(* CODESYS project SNDLTN_Hestia.library
   Company: Sandolution
   Title: SNDLTN_Hestia
   Description: Library in to aid setting up an automated domotica system.
   Author: S. Verbeek
   Version: 1.1.200929

Project tree, tasks and I/O mapping:
  libraries: StringUtils, * (System); Standard, * (System); CAA Real Time Clock Extern, * (CAA Technical Workgroup); SysSocket, * (System); CAA Net Base Services, * (CAA Technical Workgroup); SysTypes Interfaces, * (System); CmpErrors Interfaces, * (System); CAA Types, 3.0.0.2 (3S - Smart Software Solutions GmbH); CAA Tick, 3.0.0.0 (3S - Smart Software Solutions GmbH)
  Constants/
    global variables Hestia_Constants
    global variables Hestia_Properties
  Enums/
    data type Hestia_eAlarmHandler_Category
    data type Hestia_eAlarmHandler_Severity
    data type Hestia_eInputMode
    data type Hestia_eWeekday
    data type Hestia_eAlarmHandler_Sorting
  Function Blocks/
    Alarms/
      function block Hestia_AlarmHandler [ST]: Main, ShiftOutput
      function block Hestia_AlarmMessager [ST]: Main
    Colors/
      function block Hestia_Fader [ST]: Main
    Heating/
      function block Hestia_TemperatureController [ST]: Main
    Time/
      function block Hestia_WeekClock [ST]: Main, CheckWeekday
      function block Hestia_TONR [ST]: Main
    Network/
      function block Hestia_Pinger [ST]: Main
    I/O-Digital/
      function block Hestia_OutputDelay [ST]: Main
      function block Hestia_OutputHistory [ST]: Main
      function block Hestia_InputClicks [ST]: Main
      function block _Hestia_Template_xInxInvert_xOut [ST]: Main
      function block Hestia_PulseWidthModulation [ST]: Main
      function block Hestia_StateFilter [ST]: Main
    I/O-Analog/
      function block Hestia_ArrayAverage [ST]: Main
      function block Hestia_SwitchPoint_Single [ST]: Main
      function block Hestia_MovingAverage [ST]: Main
  Structs/
    data type Hestia_scWeekClockEntry
    data type Hestia_scAlarmHandler_Entry
  Variables/
  Visualizations/
  text list GlobalTextList
  program ChangeLog [ST]
  Functions/
    function Hestia_DateToWeekday [ST]
    function Hestia_ReplaceChars [ST]
    function Hestia_RandomValue [ST]
*)

// Enums/Hestia_eAlarmHandler_Category
{attribute 'qualified_only'}
{attribute 'strict'}
{attribute 'to_string'}
TYPE Hestia_eAlarmHandler_Category :
(
	System := 0,
	Security,
	Network,
	Weather,
	Climate,
	Devices,
	Monitoring
);
END_TYPE

// Enums/Hestia_eAlarmHandler_Severity
{attribute 'qualified_only'}
{attribute 'to_string'}
TYPE Hestia_eAlarmHandler_Severity :
(
	_0_Debug := 0,			//Debugging output - use only for debugging
	_1_Informational,		//Normal info for user - not important
	_2_Notice,				//Important info for user 
	_3_Warning,				 //Warning occured - attention required
	_4_Error,				//Error occured, continue processing - attention required
	_5_Critical,			//Cricital error which could comprimise functionality - action required
	_6_Alert,				//Inmediate action required to prevent further damage
	_7_Emergency			//System unusable / panic
);
END_TYPE

// Structs/Hestia_scWeekClockEntry
TYPE Hestia_scWeekClockEntry :
STRUCT
	//Week
	eWeekday					: Hestia_eWeekday;	//Individual bits also usable
	
	//Time on which output is on
	todSwitchPoint_On			: TIME_OF_DAY;		//On
	todSwitchPoint_Off			: TIME_OF_DAY;		//Off
	
	//Custom
	dwCustomAction				: DWORD;			//Specify your own custom action here, defined as number
END_STRUCT
END_TYPE

// Enums/Hestia_eInputMode
{attribute 'qualified_only'}
{attribute 'strict'}
TYPE Hestia_eInputMode :
(
	STATE := 0,
	RISING_EDGE,
	FALLING_EDGE
);
END_TYPE

// Enums/Hestia_eWeekday
{attribute 'qualified_only'}
{attribute 'to_string'}
TYPE Hestia_eWeekday :
(
	Sunday := 1,
	Monday := 2,
	Tuesday := 4,
	Wednesday := 8,
	Thursday := 16,
	Friday := 32,
	Saturday := 64,
	MonTueWedThuFri := 62,
	SatSun := 65,
	All	:= 127
) WORD;	//Set type WORD
END_TYPE

// Structs/Hestia_scAlarmHandler_Entry
TYPE Hestia_scAlarmHandler_Entry :
STRUCT
	xActive			:BOOL;
	xAckNeeded		:BOOL;
	wErrorCode		:WORD;
	eSeverity		:Hestia_eAlarmHandler_Severity;
	eCategory		:Hestia_eAlarmHandler_Category;
	sText			:STRING(Hestia_Properties.uiAlarmHandler_StringSize) := '';
END_STRUCT
END_TYPE

// Enums/Hestia_eAlarmHandler_Sorting
{attribute 'qualified_only'}
{attribute 'strict'}
TYPE Hestia_eAlarmHandler_Sorting :
(
	NoSorting := 0,
	Severity,
	TimeStamp_Oldest,
	TimeStamp_Newest
);
END_TYPE

// Constants/Hestia_Constants
{attribute 'qualified_only'}
VAR_GLOBAL CONSTANT
	uiAlarmHandler_Severity	: UINT := 8; //(0-7)
END_VAR

// Constants/Hestia_Properties
{attribute 'qualified_only'}
{attribute 'strict'}
VAR_GLOBAL CONSTANT
	uiAlarmHandler_Inputs					: UINT := 64;
	uiAlarmHandler_StringSize				: UINT := 128;
	uiAlarmHandler_Outputs					: UINT := 8;

	uiWeekClock_Entries						: UINT := 8;
	
	uiReplaceChars_StringSize				: UINT := 128;
	
	uiPinger_Samples						: UINT := 4;
	
	uiStateFilter_Inputs					: UINT := 8;
END_VAR

// ChangeLog
PROGRAM ChangeLog
VAR
END_VAR

//Library in extension to SNDLTN_Domoticz library.
//Contains functions for setting up a domotics system.

//V1.1.200929
//Fixed small bug in Switchpoint Single where hysteresis didn't work when inverted.
//Added PulseWidthModulation to control outputs.

//V1.1.200612
//Added Hestia_Pinger for ICMP pinging of network slaves
//Adjusted Hestia_ReplaceChars so it supports up to 8 chars instead of 1

//V1.1.200226
//Rewrote AlarmHandler for better sorting and handling of alarms.
//Added implementation of AlarmNotifier to send messages from the alarm handler
//Fixed bug in WeekClock on which wrong day was used for setpoints on/off spread across two days.

//V1.1.200125
//Upgraded to CoDeSys verison 3.5.14.40.
//Changed HeatingControl to TemperatureControl.

//V1.1.191207
//Added implementation of WeekClock.
//Added hysteresis to HeatingControl

//V1.1.191101:
//Added HeatingControl for simple control of heating systems.

//V1.1 - Okt 2019:
//Extension of OutputDelay and OutputHistory with eInputMode to select behaviour for different sensor types.
//Fixed bug of ColorFade where wrong constant was used. Also changed implementation to use 1..Constant instead of 0..Constant-1.

//V1.0 - Aug 2019:
//Implementation of AlarmHandler, InputClicks, OutputDelay, OutputHistory and ArrayAverage
//Sep 2019:
//Implementation of ColorFade

END_PROGRAM

// Function Blocks/Network/Hestia_Pinger
{attribute 'conditionalshow_all_locals'}
FUNCTION_BLOCK Hestia_Pinger
VAR_INPUT
	sIPAdress			:STRING := '192.168.1.1';
	udTimeOut			:UDINT := 100;
END_VAR             	 
VAR_OUTPUT          	 
	xAlive				:BOOL;
	udReplyTime			:UDINT;
END_VAR             	 
VAR                 	 
	ascResult			:ARRAY[1..Hestia_Properties.uiPinger_Samples] OF RTS_IEC_RESULT;
	rAlive_avg			:REAL;
	audReplyTime		:ARRAY[1..Hestia_Properties.uiPinger_Samples] OF UDINT;
	rReplyTime_avg		:REAL;
	SysException		:__SYSTEM.ExceptionCode;
	uiSamplesTaken		:UINT;
	idx					:INT;
END_VAR

Main();

ACTION Main:
{attribute 'conditionalshow'}
__TRY
	uiSamplesTaken := 1;
	
	IF Hestia_Properties.uiPinger_Samples > 0 THEN
		//Take all samples
		WHILE uiSamplesTaken <= Hestia_Properties.uiPinger_Samples DO
			//Get result and put in array
			ascResult[uiSamplesTaken] := SysSockPing(szIPAddress:= sIPAdress, ulTimeout:= udTimeOut, pulReplyTime:= ADR(audReplyTime[uiSamplesTaken]));
			
			//Go to next sample
			uiSamplesTaken := uiSamplesTaken + 1;
		
		END_WHILE
		
		rAlive_avg := 0;
		rReplyTime_avg := 0;
		
		FOR idx := 1 TO TO_INT(Hestia_Properties.uiPinger_Samples) DO
			//Only count valid responds, all other means offline (ERR_TIMEOUT)
			IF ascResult[idx] = CmpErrors.Errors.ERR_OK THEN
				rAlive_avg := rAlive_avg + 1;
			END_IF
			
			//Add timeout
			rReplyTime_avg := rReplyTime_avg + TO_REAL(audReplyTime[idx]);

		END_FOR
		
		//Calculate averages
		xAlive := (rAlive_avg/Hestia_Properties.uiPinger_Samples) > 0;	//One of the samples is set to true
		udReplyTime := TO_UDINT(rReplyTime_avg/Hestia_Properties.uiPinger_Samples);
		
	END_IF
	
__CATCH(SysException)
	;
__ENDTRY
END_ACTION

END_FUNCTION_BLOCK

// Functions/Hestia_ReplaceChars
FUNCTION Hestia_ReplaceChars : STRING(Hestia_Properties.uiReplaceChars_StringSize);
VAR_INPUT
	sInput			: STRING(Hestia_Properties.uiReplaceChars_StringSize);
	sCharFind		: STRING(16);
	sCharReplace	: STRING(16);
END_VAR
VAR
	iSearchPos		: INT;
	iReplaceFind	: INT;	//Check if replace string contains find string
	idx				: WORD;
END_VAR

IF sInput <> ''
AND sCharFind <> '' THEN
//AND sCharReplace <> '' THEN
	iSearchPos := 0;
	Hestia_ReplaceChars := sInput;
	
	iReplaceFind := StrFindA( ADR(sCharReplace),							//pst1
							ADR(sCharFind),									//pst2
							0);												//uiSearchStart

	FOR idx := 0 TO Hestia_Properties.uiReplaceChars_StringSize DO
		iSearchPos := StrFindA( ADR(Hestia_ReplaceChars),					//pst1
								ADR(sCharFind),								//pst2
								TO_UINT(iSearchPos));						//uiSearchStart
	
		IF iSearchPos <> 0 THEN						
			StrReplaceA(ADR(Hestia_ReplaceChars),							//pstInput
						SIZEOF(Hestia_ReplaceChars),						//uiInputBufferSize
						ADR(sCharReplace),									//pstReplaceWith
						LEN(Hestia_ReplaceChars),							//iLengthInput
						LEN(sCharFind),										//iLengthToReplace
						LEN(sCharReplace),									//iLengthToReplaceWith
						iSearchPos);										//iPosition
			iSearchPos := iSearchPos + iReplaceFind;
		ELSE
			EXIT;
		END_IF
	END_FOR
	
END_IF

END_FUNCTION

// Function Blocks/I/O-Digital/Hestia_OutputDelay
{attribute 'conditionalshow_all_locals'}
//Delay an output signal by x time
//Individual outputs are set active after set time and are reset again after the set time has passed.
//For example: 1 minut output is set after 1 minute high signal, and reset 1 minute after low signal.
FUNCTION_BLOCK Hestia_OutputDelay EXTENDS _Hestia_Template_xInxInvert_xOut
VAR_OUTPUT
	xOut_1, xOut_5, xOut_15, xOut_30, xOut_60		:BOOL;	//Input status 1/5/15/30/60m ago
END_VAR
VAR
	TON_1M, TON_5M, TON_15M, TON_30M, TON_60M		:TON;
	TOF_1M, TOF_5M, TOF_15M, TOF_30M, TOF_60M		:TOF;
END_VAR

Main();

ACTION Main:
{attribute 'conditionalshow'}
//Call parent
SUPER^.Main();

//Timed outputs
TON_1M(	IN:=xIn_int OR TOF_1M.Q, PT:=T#1M);
TOF_1M(	IN:=xIn_int AND TON_1M.Q, PT:=T#1M);
xOut_1 := TON_1M.Q OR TOF_1M.Q;

TON_5M(	IN:=xIn_int OR TOF_5M.Q, PT:=T#5M);
TOF_5M(	IN:=xIn_int AND TON_5M.Q, PT:=T#5M);
xOut_5 := TON_5M.Q OR TOF_5M.Q; 

TON_15M(IN:=xIn_int OR TOF_15M.Q, PT:=T#15M);
TOF_15M(IN:=xIn_int AND TON_15M.Q, PT:=T#15M);
xOut_15 := TON_15M.Q OR TOF_15M.Q; 

TON_30M(IN:=xIn_int OR TOF_30M.Q, PT:=T#30M);
TOF_30M(IN:=xIn_int AND TON_30M.Q, PT:=T#30M);
xOut_30 := TON_30M.Q OR TOF_30M.Q; 

TON_60M(IN:=xIn_int OR TOF_60M.Q, PT:=T#60M);
TOF_60M(IN:=xIn_int AND TON_60M.Q, PT:=T#60M);
xOut_60 := TON_60M.Q OR TOF_60M.Q;
END_ACTION

END_FUNCTION_BLOCK

// Function Blocks/I/O-Digital/_Hestia_Template_xInxInvert_xOut
{attribute 'conditionalshow'}
FUNCTION_BLOCK _Hestia_Template_xInxInvert_xOut
VAR_INPUT
	xIn			:BOOL;		//Input signal
	xInvert		:BOOL;		//Normally open / normally closed input
END_VAR
VAR_OUTPUT
	xOut		:BOOL;		//Direct output
END_VAR
VAR
	xIn_int		:BOOL;
END_VAR

//Main is called from extended slaves

ACTION Main:
//Input
xIn_int := xIn XOR xInvert;

//Direct output
xOut := xIn_int;
END_ACTION

END_FUNCTION_BLOCK

// Function Blocks/I/O-Digital/Hestia_OutputHistory
{attribute 'conditionalshow_all_locals'}
FUNCTION_BLOCK Hestia_OutputHistory EXTENDS _Hestia_Template_xInxInvert_xOut
VAR_INPUT
	eInputMode	:Hestia_eInputMode;		//Type of reaction to input
END_VAR
VAR_OUTPUT
	xOut_1, xOut_5, xOut_15, xOut_30, xOut_60		:BOOL;	//Input status 1/5/15/30/60m ago
END_VAR
VAR
	TOF_1M, TOF_5M, TOF_15M, TOF_30M, TOF_60M		:TOF;
	xIn_mode,xIn_old:BOOL;
END_VAR

Main();

ACTION Main:
{attribute 'conditionalshow'}
//Call parent
SUPER^.Main();

CASE eInputMode OF
	Hestia_eInputMode.STATE:	
		xIn_mode := xIn_int;
	
	Hestia_eInputMode.RISING_EDGE:	
		xIn_mode := xIn_int AND NOT xIn_old;
			
	Hestia_eInputMode.FALLING_EDGE:	
		xIn_mode := NOT xIn_int AND xIn_old;
END_CASE

//Save state
xIn_old := xIn_int;

//Timed outputs
TOF_1M(	IN:=xIn_mode, PT:=T#1M, Q => xOut_1);
TOF_5M(	IN:=xIn_mode, PT:=T#5M, Q => xOut_5);
TOF_15M(IN:=xIn_mode, PT:=T#15M, Q => xOut_15);
TOF_30M(IN:=xIn_mode, PT:=T#30M, Q => xOut_30);
TOF_60M(IN:=xIn_mode, PT:=T#60M, Q => xOut_60);
END_ACTION

END_FUNCTION_BLOCK

// Function Blocks/I/O-Digital/Hestia_InputClicks
{attribute 'conditionalshow_all_locals'}
FUNCTION_BLOCK Hestia_InputClicks EXTENDS _Hestia_Template_xInxInvert_xOut
VAR_INPUT
	tDebounce			:TIME := T#25MS;		//Debounce time
	tReset				:TIME := T#500MS;		//Reset outputs after set time
END_VAR
VAR_OUTPUT
	xOut_Pulse			:BOOL;
	xOut_PulseInv		:BOOL;
	xOut_Long			:BOOL;
	xOut_Single			:BOOL;
	xOut_Double			:BOOL;
	xOut_Triple			:BOOL;
END_VAR
VAR
	TON_Debounce		:TON;			//Filter input signal
	RTRIG_In			:R_TRIG;		//Pulse trigger
	FTRIG_In			:F_TRIG;		//Pulse trigger
	byCount				:BYTE;			//Count edges
	TON_Reset			:TON;			//Reset after time passed
END_VAR

Main();

ACTION Main:
{attribute 'conditionalshow'}
//Call parent
SUPER^.Main();

//Trigger on input
TON_Debounce(IN:=xIn_int, PT:=tDebounce);
RTRIG_In(CLK:=TON_Debounce.Q);
FTRIG_In(CLK:=TON_Debounce.Q);

//Count inputs
IF RTRIG_In.Q THEN
	byCount := byCount + 1;
END_IF

//Reset after set time, but reset timer each time input is received
TON_Reset(IN:=(byCount>0) AND NOT RTRIG_In.Q, PT:=tReset);
IF TON_Reset.Q AND NOT TON_Debounce.Q THEN
	byCount := 0;
END_IF

//Outputs
//xOut is written in template function 
xOut_Pulse 		:= RTRIG_In.Q;		//Single flank
xOut_PulseInv 	:= FTRIG_In.Q;		//Single flank inverted
xOut_Long 		:= TON_Debounce.Q AND TON_Reset.Q;	//Long press
xOut_Single 	:= (byCount = 1);	//1
xOut_Double 	:= (byCount = 2);	//2
xOut_Triple 	:= (byCount = 3);	//3
END_ACTION

END_FUNCTION_BLOCK

// Function Blocks/I/O-Analog/Hestia_ArrayAverage
{attribute 'conditionalshow_all_locals'}
FUNCTION_BLOCK Hestia_ArrayAverage
VAR_INPUT
	arValues		:ARRAY[1..iSamples] OF REAL := [iSamples(-999)];
END_VAR
VAR_OUTPUT
	rValue_AVG		:REAL;
END_VAR
VAR
	byX				:BYTE;
	byCnt			:BYTE;
END_VAR
VAR CONSTANT
	iSamples		:INT := 8;
END_VAR

Main();

ACTION Main:
{attribute 'conditionalshow'}
//Reset
rValue_AVG := 0;
byCnt := 0;

//Valid values
//Add all values
FOR byX := 1 TO TO_BYTE(iSamples) DO
	IF arValues[byX] <> -999 THEN
		byCnt := byCnt + 1;
		rValue_AVG := rValue_AVG + arValues[byX];
	END_IF
END_FOR

//Calc average
IF byCnt <> 0 THEN
	rValue_AVG := rValue_AVG / byCnt;
ELSE
	rValue_AVG := 0.0;
END_IF
END_ACTION

END_FUNCTION_BLOCK

// Function Blocks/Heating/Hestia_TemperatureController
{attribute 'conditionalshow_all_locals'}
FUNCTION_BLOCK Hestia_TemperatureController
VAR_INPUT
	
	rTemperature_Actual		:REAL;			//Actual room temperature (might be altered by other functions already)
	rTemperature_Hysteresis :REAL;			//Hysteresis
	
	rTemperature_Setpoint	:REAL;			//Setpoint for control
	
	xOverride				:BOOL;			//Overrule setpoint + hysteresis
	rTemperature_Override	:REAL;			//Temperature override
                             
END_VAR                      
VAR_OUTPUT	 
	xCooling				:BOOL;			//Cooling should be activate                
	xHeating				:BOOL;			//Heating should be activate
	rTemperature_Out		:REAL;			//System setpoint
END_VAR                      
VAR                          
	xActBelowHysteresis		:BOOL;
	xActAboveHysteresis		:BOOL;
END_VAR

//Call main function
Main();

ACTION Main:
{attribute 'conditionalshow'}

//Below upper hysteresis limit
//Passing from below lower hysteresis limit
IF rTemperature_Actual < rTemperature_Setpoint
AND NOT xActAboveHysteresis
AND xActBelowHysteresis THEN
	xCooling := FALSE;
	xHeating := TRUE;

//Above upper hysteresis limit
ELSIF rTemperature_Actual >= rTemperature_Setpoint THEN
	xActAboveHysteresis := TRUE;
	xActBelowHysteresis := FALSE;
	xCooling := TRUE;
	xHeating := FALSE;

//Above lower hysteresis limit
//Passing from above higher hysteresis limit
ELSIF rTemperature_Actual >= (rTemperature_Setpoint - rTemperature_Hysteresis)
AND xActAboveHysteresis
AND NOT xActBelowHysteresis THEN
	xCooling := TRUE;
	xHeating := FALSE;
	
//Below lower hysteresis limit
ELSIF rTemperature_Actual < (rTemperature_Setpoint - rTemperature_Hysteresis) THEN
	xActAboveHysteresis := FALSE;
	xActBelowHysteresis := TRUE;
	xCooling := FALSE;
	xHeating := FALSE;

//Catch
ELSE
	xCooling := FALSE;
	xHeating := FALSE;	
END_IF
	
//Override active
IF xOverride THEN
	rTemperature_Out := rTemperature_Override;	
//Normal operation
ELSE
	rTemperature_Out := rTemperature_Setpoint;
END_IF
END_ACTION

END_FUNCTION_BLOCK

// Functions/Hestia_DateToWeekday
{attribute 'conditionalshow_all_locals'}
FUNCTION Hestia_DateToWeekday : Hestia_eWeekday
VAR_INPUT
	dDate				:DATE;	//Date to convert
END_VAR 
VAR
	sDate				:STRING(12);
	iYear,iMonth,iDay	:INT;
	iYearDigit,iCentury	:INT;
	iCalculate			:INT;
END_VAR

//Conversion is done using the Key Value method

//Convert to STRING and get INT values
sDate 		:= TO_STRING(dDate);
iYear 		:= TO_INT(MID(sDate,4,3));	//Extract length 4 from pos 3 (1970)
iYearDigit 	:= TO_INT(MID(sDate,2,5));	//Extract length 2 from pos 5 (70)
iCentury 	:= TO_INT(MID(sDate,2,3));	//Extract length 2 from pos 3 (19)
iMonth 		:= TO_INT(MID(sDate,2,8));	//Extract length 2 from pos 8 (01)
iDay 		:= TO_INT(MID(sDate,2,11));	//Extract length 2 from pos 11 (01)

//Take last two digits of the year and divide by 4, drop remainder
iCalculate 	:= iYearDigit / 4;
//Add day of month
iCalculate 	:=  iCalculate + iDay;
//Add key value
CASE iMonth OF
	1:	iCalculate := iCalculate + 1;
	2:	iCalculate := iCalculate + 4;
	3:	iCalculate := iCalculate + 4;
	4:	iCalculate := iCalculate + 0;
	5:	iCalculate := iCalculate + 2;
	6:	iCalculate := iCalculate + 5;
	7:	iCalculate := iCalculate + 0;
	8:	iCalculate := iCalculate + 3;
	9:	iCalculate := iCalculate + 6;
	10:	iCalculate := iCalculate + 1;
	11:	iCalculate := iCalculate + 4;
	12:	iCalculate := iCalculate + 6;
END_CASE
//Substract 1 for Jan/Feb if leap year
IF ((iYear MOD 4) = 0) AND (iMonth = 1 OR iMonth = 2) THEN
	iCalculate := iCalculate - 1;
END_IF
//Add century code
//Note that this only works from 1900 to 2100, date type doesn't support other centuries
CASE iCentury OF
	19:	iCalculate := iCalculate + 0;
	20:	iCalculate := iCalculate + 6;
	21:	iCalculate := iCalculate + 4;
END_CASE
//Add year digits
iCalculate := iCalculate + iYearDigit;
//Devide by 7 and take remainder
iCalculate := iCalculate MOD 7;
//Fix if 0, this is also saturday
IF iCalculate = 0 THEN
	iCalculate := 7;
END_IF
//Output
Hestia_DateToWeekday := TO_WORD(iCalculate);

END_FUNCTION

// Function Blocks/Time/Hestia_WeekClock
{attribute 'conditionalshow_all_locals'}
FUNCTION_BLOCK Hestia_WeekClock
VAR_INPUT
	xEnable					: BOOL;
	dtActDateTime			: DATE_AND_TIME;
	ascWeekClock_Entries	: ARRAY[1..Hestia_Properties.uiWeekClock_Entries] OF Hestia_scWeekClockEntry;
END_VAR
VAR_OUTPUT
	byEntryActive			: BYTE;
	dwAction				: DWORD;
END_VAR
VAR
	idx						: WORD;
	axSaveNextDay			: ARRAY[1..Hestia_Properties.uiWeekClock_Entries] OF BOOL;
END_VAR

Main();

ACTION Main:
{attribute 'conditionalshow'}

//Reset outputs
byEntryActive := 0;
dwAction := 0;

IF xEnable THEN
	
	//Loop all entries
	FOR idx := 1 TO Hestia_Properties.uiWeekClock_Entries DO
		
		//Check if entries are valid
		IF ascWeekClock_Entries[idx].todSwitchPoint_On <> TOD#00:00:00
		AND ascWeekClock_Entries[idx].todSwitchPoint_Off <> TOD#00:00:00
		AND ascWeekClock_Entries[idx].todSwitchPoint_On <> ascWeekClock_Entries[idx].todSwitchPoint_Off THEN
		
			//Time on/off lays in the same day and in correct order
			IF ascWeekClock_Entries[idx].todSwitchPoint_On < ascWeekClock_Entries[idx].todSwitchPoint_Off THEN
			
				//Actual time within range of setpoints
				IF TO_TOD(dtActDateTime) >= ascWeekClock_Entries[idx].todSwitchPoint_On
				AND TO_TOD(dtActDateTime) < ascWeekClock_Entries[idx].todSwitchPoint_Off
				//Correct day active
				AND CheckWeekday(TO_DATE(dtActDateTime), ascWeekClock_Entries[idx].eWeekday, FALSE) THEN
					byEntryActive := TO_BYTE(idx);
					dwAction := ascWeekClock_Entries[idx].dwCustomAction;
				END_IF	
				
			//Time on/off lay on two different days. Use weekday of ON switchpoint
			ELSIF ascWeekClock_Entries[idx].todSwitchPoint_On > ascWeekClock_Entries[idx].todSwitchPoint_Off THEN
				//Actual time within range of setpoints
				IF (TO_TOD(dtActDateTime) >= ascWeekClock_Entries[idx].todSwitchPoint_On
					OR (TO_TOD(dtActDateTime) < ascWeekClock_Entries[idx].todSwitchPoint_Off AND axSaveNextDay[idx]))
				AND (TO_TOD(dtActDateTime) < ascWeekClock_Entries[idx].todSwitchPoint_Off 
					OR (TO_TOD(dtActDateTime) >= ascWeekClock_Entries[idx].todSwitchPoint_On AND (TO_TOD(dtActDateTime) <= TOD#23:59:59)))
				//Correct day active
				AND (CheckWeekday(TO_DATE(dtActDateTime), ascWeekClock_Entries[idx].eWeekday, TRUE) OR axSaveNextDay[idx]) THEN
					axSaveNextDay[idx] := TRUE;
					byEntryActive := TO_BYTE(idx);
					dwAction := ascWeekClock_Entries[idx].dwCustomAction;
				ELSE
					axSaveNextDay[idx] := FALSE;
				END_IF	
			END_IF
			
		END_IF
	
	END_FOR

END_IF
END_ACTION

METHOD CheckWeekday : BOOL
VAR_INPUT
	dActDate	: DATE;
	eWeekday	: Hestia_eWeekday;
	xDayInPast	: BOOL;
END_VAR
CheckWeekday := 
			//Check current day (setpoints on same day)
			(NOT xDayInPast
			AND ((Hestia_DateToWeekday(dActDate) = 1 AND eWeekday.0)
			OR (Hestia_DateToWeekday(dActDate) = 2 AND eWeekday.1)
			OR (Hestia_DateToWeekday(dActDate) = 3 AND eWeekday.2)
			OR (Hestia_DateToWeekday(dActDate) = 4 AND eWeekday.3)
			OR (Hestia_DateToWeekday(dActDate) = 5 AND eWeekday.4)
			OR (Hestia_DateToWeekday(dActDate) = 6 AND eWeekday.5)
			OR (Hestia_DateToWeekday(dActDate) = 7 AND eWeekday.6)))
			
			//Check previous day (setpoints on/off on different days)
			OR (xDayInPast
			AND ((Hestia_DateToWeekday(dActDate) = 1 AND eWeekday.1)
			OR (Hestia_DateToWeekday(dActDate) = 2 AND eWeekday.2)
			OR (Hestia_DateToWeekday(dActDate) = 3 AND eWeekday.3)
			OR (Hestia_DateToWeekday(dActDate) = 4 AND eWeekday.4)
			OR (Hestia_DateToWeekday(dActDate) = 5 AND eWeekday.5)
			OR (Hestia_DateToWeekday(dActDate) = 6 AND eWeekday.6)
			OR (Hestia_DateToWeekday(dActDate) = 7 AND eWeekday.0)));
END_METHOD

END_FUNCTION_BLOCK

// Function Blocks/Alarms/Hestia_AlarmHandler
{attribute 'conditionalshow_all_locals'}
FUNCTION_BLOCK Hestia_AlarmHandler
VAR_INPUT
	xEnable				:BOOL;
	dtCurrentDateTime	:DT;
	ascLogEntries		:ARRAY[1..Hestia_Properties.uiAlarmHandler_Inputs] OF Hestia_scAlarmHandler_Entry;
	eSortingMode		:Hestia_eAlarmHandler_Sorting;
END_VAR
VAR_OUTPUT
	ascLogOutput		:ARRAY[1..Hestia_Properties.uiAlarmHandler_Outputs] OF Hestia_scAlarmHandler_Entry;
	adtLogOutput		:ARRAY[1..Hestia_Properties.uiAlarmHandler_Outputs] OF DT;
END_VAR
VAR
	adtLogEntries		:ARRAY[1..Hestia_Properties.uiAlarmHandler_Inputs] OF DT;
	axLogEntries_Mem	:ARRAY[1..Hestia_Properties.uiAlarmHandler_Inputs] OF BOOL;
	
	iFor_Entries		:INT;
	iFor_Output			:INT;
	iFor_Severity		:INT;
	iFor_TimeStamp		:INT;
	uiLogOutput_Index	:UINT;
	
	scDefaultEntry		:Hestia_scAlarmHandler_Entry;
	
END_VAR

Main();

ACTION Main:
{attribute 'conditionalshow'}

IF xEnable THEN

	//Clock timestamp for all entries
	FOR iFor_Entries := 1 TO TO_INT(Hestia_Properties.uiAlarmHandler_Inputs) BY 1 DO
		IF ascLogEntries[iFor_Entries].xActive 
		AND NOT axLogEntries_Mem[iFor_Entries] THEN
			adtLogEntries[iFor_Entries] := dtCurrentDateTime;
			axLogEntries_Mem[iFor_Entries] := TRUE;
		ELSIF NOT ascLogEntries[iFor_Entries].xActive THEN
			adtLogEntries[iFor_Entries] := DT#1970-1-1-0:0:0;
			axLogEntries_Mem[iFor_Entries] := FALSE;
		END_IF
	END_FOR
	
	
	//Output in order of severity
	IF eSortingMode = Hestia_eAlarmHandler_Sorting.Severity THEN
		uiLogOutput_Index := 1;
		FOR iFor_Severity := TO_INT(Hestia_Constants.uiAlarmHandler_Severity-1) TO 0 BY -1 DO		//Loop all severity from 7 to 0
			FOR iFor_Entries := 1 TO TO_INT(Hestia_Properties.uiAlarmHandler_Inputs) BY 1 DO		//Loop all input entries
				IF ascLogEntries[iFor_Entries].eSeverity = iFor_Severity							//Check if severity is eqal 
				AND ascLogEntries[iFor_Entries].xActive												//Check if alarm is active
				AND uiLogOutput_Index <= Hestia_Properties.uiAlarmHandler_Outputs THEN				//Check if within range of output
					ascLogOutput[uiLogOutput_Index] := ascLogEntries[iFor_Entries];					//Output entry
					adtLogOutput[uiLogOutput_Index] := adtLogEntries[iFor_Entries];					//Output datetime
					uiLogOutput_Index := uiLogOutput_Index + 1;										//Next output
				ELSIF uiLogOutput_Index > Hestia_Properties.uiAlarmHandler_Outputs THEN				//Done, output full
					EXIT;
				END_IF
			END_FOR
		END_FOR
		
	//Output timestamp oldest to newest
	ELSIF eSortingMode = Hestia_eAlarmHandler_Sorting.TimeStamp_Oldest THEN
		
		FOR iFor_Entries := 1 TO TO_INT(Hestia_Properties.uiAlarmHandler_Outputs) BY 1 DO			//Reset array
			ascLogOutput[iFor_Entries] := scDefaultEntry;
			adtLogOutput[iFor_Entries] := DT#1970-1-1-0:0:0;
		END_FOR
	
		uiLogOutput_Index := 1;
		FOR iFor_Entries := 1 TO TO_INT(Hestia_Properties.uiAlarmHandler_Inputs) BY 1 DO			//Loop all input entries
			IF ascLogEntries[iFor_Entries].xActive THEN												//Check if alarm is active
				FOR iFor_TimeStamp := 1 TO TO_INT(Hestia_Properties.uiAlarmHandler_Outputs) BY 1 DO	//Check with all elements of output
					IF adtLogOutput[iFor_TimeStamp] <> DT#1970-01-01-00:00:00						//Entry is not empty
					AND adtLogEntries[iFor_Entries] <= adtLogOutput[iFor_TimeStamp] THEN			//Entry is older (or equal) than output
						IF iFor_TimeStamp < 8 THEN
							ShiftOutput(uiPosition:=TO_UINT(iFor_TimeStamp), xInvert:=FALSE);		//Shift output array upwards
						END_IF
						ascLogOutput[iFor_TimeStamp] := ascLogEntries[iFor_Entries];				//Output entry
						adtLogOutput[iFor_TimeStamp] := adtLogEntries[iFor_Entries];				//Output datetime
						uiLogOutput_Index := uiLogOutput_Index + 1;									//Next output
						EXIT;
					ELSIF adtLogOutput[iFor_TimeStamp] = DT#1970-01-01-00:00:00 					//Entry empty
					AND uiLogOutput_Index <= Hestia_Properties.uiAlarmHandler_Outputs THEN			//Check if within range of output
						ascLogOutput[uiLogOutput_Index] := ascLogEntries[iFor_Entries];				//Output entry
						adtLogOutput[uiLogOutput_Index] := adtLogEntries[iFor_Entries];				//Output datetime
						uiLogOutput_Index := uiLogOutput_Index + 1;									//Next output
						EXIT;
					END_IF
				END_FOR
			END_IF
		END_FOR
		
	//Just output in order of entry
	ELSIF eSortingMode = Hestia_eAlarmHandler_Sorting.NoSorting THEN
		uiLogOutput_Index := 1;
		FOR iFor_Entries := 1 TO TO_INT(Hestia_Properties.uiAlarmHandler_Inputs) BY 1 DO			//Loop all input entries
			IF ascLogEntries[iFor_Entries].xActive													//Check if alarm is active
			AND uiLogOutput_Index <= Hestia_Properties.uiAlarmHandler_Outputs THEN					//Check if within range of output
				ascLogOutput[uiLogOutput_Index] := ascLogEntries[iFor_Entries];						//Output entry
				adtLogOutput[uiLogOutput_Index] := adtLogEntries[iFor_Entries];						//Output datetime
				uiLogOutput_Index := uiLogOutput_Index + 1;											//Next output
			ELSIF uiLogOutput_Index > Hestia_Properties.uiAlarmHandler_Outputs THEN					//Done, output full
				EXIT;
			END_IF
		END_FOR
	END_IF
	
	//Delete old data
	IF uiLogOutput_Index < Hestia_Properties.uiAlarmHandler_Outputs THEN
		FOR iFor_Output := TO_INT(uiLogOutput_Index) TO TO_INT(Hestia_Properties.uiAlarmHandler_Outputs) BY 1 DO
			ascLogOutput[iFor_Output] := scDefaultEntry;
			adtLogOutput[iFor_Output] := DT#1970-1-1-0:0:0;
		END_FOR
	END_IF

//Not enabled
ELSE
	//Delete all data
	FOR iFor_Output := 1 TO TO_INT(Hestia_Properties.uiAlarmHandler_Outputs) BY 1 DO
		ascLogOutput[iFor_Output] := scDefaultEntry;
		adtLogOutput[iFor_Output] := DT#1970-1-1-0:0:0;
	END_FOR
END_IF
END_ACTION

METHOD INTERNAL ShiftOutput
VAR_INPUT
	uiPosition		: UINT;
	xInvert			: BOOL;
END_VAR
VAR
	iForLoop		: INT;
END_VAR
IF NOT xInvert
AND uiPosition > 1
AND uiPosition < Hestia_Properties.uiAlarmHandler_Outputs THEN
	FOR iForLoop := TO_INT(Hestia_Properties.uiAlarmHandler_Outputs) TO MAX(TO_INT(uiPosition),2) BY -1 DO
		ascLogOutput[iForLoop] := ascLogOutput[iForLoop-1];
		adtLogOutput[iForLoop] := adtLogOutput[iForLoop-1];
	END_FOR
ELSIF xInvert
AND uiPosition <= Hestia_Properties.uiAlarmHandler_Outputs THEN
	FOR iForLoop :=  TO_INT(uiPosition) TO TO_INT(Hestia_Properties.uiAlarmHandler_Outputs-1) BY 1 DO
		ascLogOutput[iForLoop] := ascLogOutput[iForLoop+1];
		adtLogOutput[iForLoop] := adtLogOutput[iForLoop+1];
	END_FOR
END_IF
END_METHOD

END_FUNCTION_BLOCK

// Function Blocks/Alarms/Hestia_AlarmMessager
{attribute 'conditionalshow_all_locals'}
FUNCTION_BLOCK Hestia_AlarmMessager
VAR_INPUT
	ascAlarmHandler_Outputs			:ARRAY[1..Hestia_Properties.uiAlarmHandler_Outputs] OF Hestia_scAlarmHandler_Entry;
	eSeverity_Minimal				:Hestia_eAlarmHandler_Severity := Hestia_eAlarmHandler_Severity._0_Debug;
	eSeverity_Maximal				:Hestia_eAlarmHandler_Severity := Hestia_eAlarmHandler_Severity._7_Emergency;
	xUseAlarmText					:BOOL;	//Use text instead of error code (error codes should be unique)
	xMessageSent					:BOOL;
END_VAR                     		
VAR_OUTPUT                  		
	ascAlarms						:ARRAY[1..Hestia_Properties.uiAlarmHandler_Outputs] OF Hestia_scAlarmHandler_Entry;
	scAlarmOutput					:Hestia_scAlarmHandler_Entry := (sText := 'NULL');
END_VAR                     	
VAR                         	
	asMessages_int					:ARRAY[1..Hestia_Properties.uiAlarmHandler_Outputs] OF STRING(Hestia_Properties.uiAlarmHandler_StringSize);
	awErrorCode_int					:ARRAY[1..Hestia_Properties.uiAlarmHandler_Outputs] OF WORD;
	
	scMessage_Empty					:Hestia_scAlarmHandler_Entry := (sText := 'NULL');
	
	wErrorCode_int					:WORD;
	
	xMessageSent_mem				:BOOL;
	xMessageSending					:BOOL;
	//Notification system to Domoticz	
	uiFor_AlarmHandler_Outputs		:UINT;  
	uiFor_Messages					:UINT;
	uiFor_Messages_int				:UINT;
	uiFor_Messages_int_EmptyPlace	:UINT;
END_VAR

Main();

ACTION Main:
{attribute 'conditionalshow'}
//Empty output array
FOR uiFor_Messages := 1 TO Hestia_Properties.uiAlarmHandler_Outputs DO
	ascAlarms[uiFor_Messages] := scMessage_Empty;
END_FOR

//Fill output array with categories
FOR uiFor_AlarmHandler_Outputs := 1 TO Hestia_Properties.uiAlarmHandler_Outputs DO	 
	//Notifications
	FOR uiFor_Messages := 1 TO Hestia_Properties.uiAlarmHandler_Outputs DO
		IF ascAlarmHandler_Outputs[uiFor_AlarmHandler_Outputs].xActive
		AND ascAlarmHandler_Outputs[uiFor_AlarmHandler_Outputs].eSeverity >= eSeverity_Minimal
		AND ascAlarmHandler_Outputs[uiFor_AlarmHandler_Outputs].eSeverity <= eSeverity_Maximal
		AND NOT ascAlarms[uiFor_Messages].xActive
		AND (ascAlarms[uiFor_Messages].sText = '' OR ascAlarms[uiFor_Messages].sText = 'NULL')
		AND ascAlarms[uiFor_Messages].wErrorCode = 0 THEN
			ascAlarms[uiFor_Messages] := ascAlarmHandler_Outputs[uiFor_AlarmHandler_Outputs];
			EXIT;
		END_IF
	END_FOR
END_FOR;


//Check if entries from list are in list send, otherwise send message and add to list
FOR uiFor_Messages := 1 TO Hestia_Properties.uiAlarmHandler_Outputs DO
	FOR uiFor_Messages_int := 1 TO Hestia_Properties.uiAlarmHandler_Outputs DO
		//Already being send
		IF ascAlarms[uiFor_Messages].sText = scAlarmOutput.sText THEN
			EXIT;
		END_IF	
		//Check if already sent
		IF NOT xMessageSending
		AND ascAlarms[uiFor_Messages].sText <> ''
		AND ((ascAlarms[uiFor_Messages].sText = asMessages_int[uiFor_Messages_int]
		AND xUseAlarmText)
		OR (ascAlarms[uiFor_Messages].wErrorCode = awErrorCode_int[uiFor_Messages_int]
		 AND NOT xUseAlarmText)) THEN
			EXIT;
		END_IF
	END_FOR
	//Array end
	IF uiFor_Messages_int >= Hestia_Properties.uiAlarmHandler_Outputs //Loop at end, send entry
	AND NOT xMessageSending
	AND ascAlarms[uiFor_Messages].sText <> '' THEN
		xMessageSending := TRUE;
		scAlarmOutput := ascAlarms[uiFor_Messages];
		wErrorCode_int := ascAlarms[uiFor_Messages].wErrorCode;
	END_IF
END_FOR
//Add to array when done
IF NOT xMessageSent_mem AND xMessageSent THEN	//Add to array if send
	FOR uiFor_Messages_int_EmptyPlace := 1 TO Hestia_Properties.uiAlarmHandler_Outputs DO	//Find place in array
		IF asMessages_int[uiFor_Messages_int_EmptyPlace] = '' THEN
			asMessages_int[uiFor_Messages_int_EmptyPlace] := scAlarmOutput.sText;
			awErrorCode_int[uiFor_Messages_int_EmptyPlace] := wErrorCode_int;
			scAlarmOutput := scMessage_Empty;
			xMessageSending := FALSE;
			EXIT;
		END_IF
	END_FOR
END_IF

//Check if entries from send list are still in original list, otherwise delete from list send
FOR uiFor_Messages_int := 1 TO Hestia_Properties.uiAlarmHandler_Outputs DO
	FOR uiFor_Messages := 1 TO Hestia_Properties.uiAlarmHandler_Outputs DO
		IF ((asMessages_int[uiFor_Messages_int] <> ''
		AND asMessages_int[uiFor_Messages_int] = ascAlarms[uiFor_Messages].sText 
		AND xUseAlarmText)
		OR (awErrorCode_int[uiFor_Messages_int] <> 0
		AND awErrorCode_int[uiFor_Messages_int] = ascAlarms[uiFor_Messages].wErrorCode 
		AND NOT xUseAlarmText)) THEN	//If exists, then exit
			EXIT;
		END_IF
	END_FOR
	//Array end
	IF uiFor_Messages >= Hestia_Properties.uiAlarmHandler_Outputs THEN	//Loop at end, delete entry
		asMessages_int[uiFor_Messages_int] := '';
		awErrorCode_int[uiFor_Messages_int] := 0;
	END_IF
END_FOR

//Store puls
xMessageSent_mem := xMessageSent;
END_ACTION

END_FUNCTION_BLOCK

// Function Blocks/I/O-Analog/Hestia_SwitchPoint_Single
FUNCTION_BLOCK Hestia_SwitchPoint_Single
VAR_INPUT
	rInput			: REAL;
	rSwitchPoint	: REAL;
	rHysteresis		: REAL;
	xInvert			: BOOL;		//Hysteresis added to value instead of substracted
END_VAR
VAR_OUTPUT
	xOut			: BOOL;
END_VAR
VAR
END_VAR

Main();

ACTION Main:
IF NOT xInvert THEN
	IF rInput >= rSwitchPoint THEN
		xOut := TRUE;
	ELSIF rInput <= (rSwitchPoint-rHysteresis) THEN
		xOut := FALSE;
	END_IF
ELSIF xInvert THEN
	IF rInput <= rSwitchPoint THEN
		xOut := TRUE;
	ELSIF rInput >= (rSwitchPoint+rHysteresis) THEN
		xOut := FALSE;
	END_IF
END_IF
END_ACTION

END_FUNCTION_BLOCK

// Functions/Hestia_RandomValue
FUNCTION Hestia_RandomValue : UDINT
VAR_INPUT
	udiLowLimit			:UDINT;		//Min number
	udiHighLimit		:UDINT;		//Max number
END_VAR
VAR
	caaTick				:CAA.TICK;
	udiTick				:UDINT;
	udiShiftL			:UDINT;
	udiShiftR			:UDINT;
	udiTickShiftL		:UDINT;
	udiTickDiv			:UDINT;
	udiTickShiftR		:UDINT;
	udiTickModulo		:UDINT;	
END_VAR

caaTick := TICKS.GetTick(0);

//16/32/64 bit system
{IF hasvalue (RegisterSize, '16')}
udiTick := UINT_TO_UDINT(caaTick);           
{ELSIF hasvalue (RegisterSize, '32')}
udiTick := caaTick;      
{ELSIF hasvalue (RegisterSize, '64')}
udiTick := ULINT_TO_UDINT(caaTick);   
{END_IF}

udiShiftL := (udiTick MOD 17) + 1;	//prime number > avoid 0
udiShiftR := (udiTick MOD 7) + 1;	//prime number > avoid 0

udiTickShiftL := SHL(udiTick, udiShiftL);
udiTickShiftR := SHR(udiTick, udiShiftR);
udiTickDiv := udiTickShiftL / udiTickShiftR;
udiTickModulo := udiTickShiftR MOD (udiHighLimit-udiLowLimit+1);
Hestia_RandomValue := udiTickModulo + udiLowLimit;

END_FUNCTION

// Function Blocks/Time/Hestia_TONR
FUNCTION_BLOCK Hestia_TONR
VAR_INPUT
	IN:BOOL;
	PT:TIME;
	RST:BOOL;
END_VAR
VAR_OUTPUT
	Q:BOOL;
	ET:TIME;
END_VAR
VAR
	F_TRIG0:F_TRIG;
	TIMER:TON;
END_VAR
VAR RETAIN
	PASSED:TIME;
END_VAR

Main();

ACTION Main:
//Reset passed time
IF RST THEN
	PASSED :=T#0S;
END_IF

//Save time on passed
F_TRIG0(CLK:= IN);
//Save time on disable
IF F_TRIG0.Q THEN
	PASSED := TIMER.ET + PASSED;
END_IF

//Protection for negative time (already passed)
IF PASSED >= PT THEN
	TIMER.PT := (T#0MS);		//Time already passed
ELSE
	TIMER.PT := (PT - PASSED);
END_IF

//Call timer
TIMER(IN:= IN AND NOT RST);

//Write output on timer output or when time has passed (double - to be sure)
Q := TIMER.Q OR (ET >= PT);

//Construct elapsed time AFTER output
IF IN THEN
	ET := TIMER.ET + PASSED;
//Disabled, PT is changed (smaller than ET)
ELSIF ET > PT THEN
	ET := PT;
	PASSED := ET;
//Disabled
ELSE
	ET := PASSED;
END_IF
END_ACTION

END_FUNCTION_BLOCK

// Function Blocks/I/O-Digital/Hestia_PulseWidthModulation
FUNCTION_BLOCK Hestia_PulseWidthModulation		//Create PWM with regular DO slice
VAR_INPUT
	rFrequency					:REAL;				//Frequency in Hz
	iPulseWidth					:INT;				//Pulse width in %
END_VAR                         
VAR_OUTPUT                      
	xOut						:BOOL;
END_VAR                         
VAR                             
	rMinFrequency				:REAL				:= 0.1;	//0.1Hz might be needed on some systems
	rMaxFrequency				:REAL				:= 120;	//Use 120Hz max, this is the max usable with a 4ms task cycle
	
	rMinPwm						:REAL				:= 1;	//Min 0%
	rMaxPwm						:REAL				:= 100;	//Max 100%
	rPwm						:REAL;
	
	tTotalTime					:TIME;
	tTimeOn						:TIME;
	tTimeOff					:TIME;
	
	TON1:						TON;
	TOF1:						TOF;
	
END_VAR

Main();

ACTION Main:
rFrequency	:= LIMIT(rMinFrequency, rFrequency, rMaxFrequency);				//Overwrite value if needed
rPwm		:= LIMIT(rMinPwm, (iPulseWidth/100.0) * rMaxPwm, rMaxPwm);		//Calculate value
            
tTotalTime	:= TO_TIME(TO_REAL(T#1S) / rFrequency);							//Get total cycle time
tTimeOn		:= TO_TIME(TO_REAL(tTotalTime) / 100 * rPwm);					//Calculate on-time
tTimeOff	:= tTotalTime - tTimeOn;										//Calculate off-time

TON1(IN:= TOF1.Q, PT:= tTimeOff, Q=> xOut);
TOF1(IN:= NOT TON1.Q, PT:= tTimeOn);
END_ACTION

END_FUNCTION_BLOCK

// Function Blocks/I/O-Analog/Hestia_MovingAverage
FUNCTION_BLOCK Hestia_MovingAverage
VAR_INPUT
	xEnable				:BOOL;		//Enable FB
	rValue				:REAL;		//Input (measured value)
	iSamples			:INT;		//Amount of measurements
	tSampleTime			:TIME;		//Time between measurements
END_VAR
VAR_OUTPUT
	xOverflow			:BOOL;		//Error 
	rValueAvg			:REAL;		//Output
END_VAR
VAR
	arSamples			:ARRAY[0..gc_iMaxSamples] OF LREAL;	//Store samples
	rValueCalc			:REAL;		//Calculate average
	iSamplesActive		:INT;		//Active samples
	idx					:INT;		//For loops
	TON_Sample			:TON;
	xSampleDone			:BOOL;		//Sample
END_VAR
VAR CONSTANT
	gc_iMaxSamples		:INT := 32;
END_VAR

Main();

ACTION Main:
//FB Enabled
IF xEnable THEN
    //Change value when setpoint is set lower
    IF iSamplesActive > iSamples THEN
        iSamplesActive := iSamples;
    END_IF;
    
    IF TON_Sample.Q AND iSamples <= gc_iMaxSamples THEN  //Add value if not outside boundry
        IF iSamplesActive < iSamples THEN        //Fill up filter until full
            arSamples[iSamplesActive + 1] := rValue;
            iSamplesActive := iSamplesActive + 1;
        ELSIF iSamplesActive >= iSamples THEN    //Shift everything left
            FOR idx := 0 TO (iSamples - 1) BY 1 DO
                arSamples[idx] := arSamples[idx + 1];
            END_FOR;
            arSamples[iSamplesActive] := rValue;
        END_IF;
        
        //Calculate average
        rValueCalc := 0;
        IF iSamplesActive > 0 THEN
            FOR idx := 1 TO iSamplesActive BY 1 DO
                rValueCalc := rValueCalc + arSamples[idx];
            END_FOR;
            rValueAvg := rValueCalc / iSamplesActive;
        END_IF;
        
        xSampleDone := TRUE;

    END_IF
    
//Dsiabled; remove all values
ELSE
    rValueAvg := 0.0;
    FOR idx := 0 TO gc_iMaxSamples DO
        arSamples[idx] := 0.0;
    END_FOR;
END_IF;

//Make pulse to sample
TON_Sample(IN := (NOT xSampleDone),
            PT := tSampleTime);
			
//Reset sample (Bit 1 cycle active)
IF xSampleDone THEN
    xSampleDone := FALSE;
END_IF;

//To much samples configured
xOverflow :=iSamples > gc_iMaxSamples;
END_ACTION

END_FUNCTION_BLOCK

// Function Blocks/Colors/Hestia_Fader
{attribute 'conditionalshow_all_locals'}
FUNCTION_BLOCK Hestia_Fader
VAR_INPUT
	xEnable					:BOOL;
	tFadeTime				:TIME := T#3S;
	uiFadeSteps				:UINT := 16;
	rValueIn				:REAL;
END_VAR
VAR_OUTPUT
	xFading					:BOOL;
	rValueOut				:REAL;
END_VAR
VAR
	rValueIn_int			:REAL;	//Store value to see if it changed
	rValueIn_mem			:REAL;	//Store value to see if it changed
	rValueSingleStep		:REAL;	//Signle step
	TON_Fade				:TON;
	xFading_int				:BOOL;
	uiFadeStepsTaken		:UINT;
END_VAR

Main();

ACTION Main:
{attribute 'conditionalshow'}

//Check if input values have changed and calculate fade parameters
IF rValueIn <> rValueIn_int THEN
	rValueSingleStep := rValueIn - rValueIn_int;	//Calculate difference
	rValueSingleStep := rValueSingleStep / uiFadeSteps;	//Divide by amount of steps
	rValueIn_int := rValueIn;	//Store value
	xFading_int := TRUE;
	uiFadeStepsTaken := 1;
END_IF

//Increase value
IF TON_Fade.Q THEN
	IF uiFadeStepsTaken < uiFadeSteps THEN
		uiFadeStepsTaken := uiFadeStepsTaken + 1;
	ELSE
		rValueIn_mem := rValueIn_int;
		xFading_int := FALSE;
	END_IF
END_IF

//Write outputs
//Status
xFading := xEnable
		AND xFading_int;

//Fading output
IF NOT xEnable THEN
	rValueOut := rValueIn;
ELSIF xFading_int THEN
	rValueOut := rValueIn_mem + (rValueSingleStep * uiFadeStepsTaken);
ELSE
	rValueOut := rValueIn_mem;	
END_IF

//Call timer
TON_Fade(
	IN:= NOT TON_Fade.Q
		AND xFading_int,
	PT:=TO_TIME(TO_UDINT(tFadeTime)/uiFadeSteps)
);
END_ACTION

END_FUNCTION_BLOCK

// Function Blocks/I/O-Digital/Hestia_StateFilter
FUNCTION_BLOCK Hestia_StateFilter
VAR_INPUT
	axInput			: ARRAY[1..Hestia_Properties.uiStateFilter_Inputs] OF BOOL;
	axInvert		: ARRAY[1..Hestia_Properties.uiStateFilter_Inputs] OF BOOL;
	aeInputMode		: ARRAY[1..Hestia_Properties.uiStateFilter_Inputs] OF Hestia_eInputMode;
END_VAR
VAR_OUTPUT
	xOutput			: BOOL;	//Any output active
	axOutput		: ARRAY[1..Hestia_Properties.uiStateFilter_Inputs] OF BOOL;
END_VAR
VAR
	axInput_int		: ARRAY[1..Hestia_Properties.uiStateFilter_Inputs] OF BOOL;
	axInput_old		: ARRAY[1..Hestia_Properties.uiStateFilter_Inputs] OF BOOL;
	idx				: WORD;
END_VAR

Main();

ACTION Main:
//Reset
xOutput := FALSE;

//Run functions
FOR idx := 1 TO Hestia_Properties.uiStateFilter_Inputs DO
	
	//Perform inversion
	axInput_int[idx] := axInput[idx] XOR axInvert[idx];

	//Select proper trigger
	CASE aeInputMode[idx] OF
	Hestia_eInputMode.STATE:	
		axOutput[idx] := axInput_int[idx];
	
	Hestia_eInputMode.RISING_EDGE:	
		axOutput[idx] := axInput_int[idx] AND NOT axInput_old[idx];
			
	Hestia_eInputMode.FALLING_EDGE:	
		axOutput[idx] := NOT axInput[idx] AND axInput_old[idx];
	END_CASE
	
	//Save state
	axInput_old[idx] := axInput_int[idx];
	
	//Set collect output
	IF axOutput[idx] THEN
		xOutput := TRUE;
	END_IF
END_FOR
END_ACTION

END_FUNCTION_BLOCK
